// TIA Portal V16 export
// export: Created 2024-09-05T17:39:11.9932458Z, ExportSetting WithDefaults, DisplayName Totally Integrated Automation Portal, DisplayVersion V16 Update 6, DisplayName TIA Portal Version Control Interface, DisplayVersion V16 Update 2, DisplayName TIA Portal Openness, DisplayVersion V16 Update 6, DisplayName STEP 7 Professional, DisplayVersion V16 Update 6, DisplayName STEP 7 Safety, DisplayVersion V16, DisplayName WinCC Advanced, DisplayVersion V16 Update 6
DATA_BLOCK "ServoMain_DB"   // DB6
VERSION : 0.1
// stored: AutoNumber true, DBAccessibleFromOPCUA true, InstanceOfName ServoMain, InstanceOfType FB
"ServoMain"
   // VAR
   //    "TO_BasicPos_TA1-3MA_Instance" { S7_SetPoint := 'True'} : TO_BasicPos;
   //    IEC_Timer_0_Instance { S7_SetPoint := 'True'} : TON_TIME;
   //    "ServoControl_TA1-3MA_Instance" { S7_SetPoint := 'True'} : "ServoControl";
   //    IEC_Timer_0_Instance_1 { S7_SetPoint := 'True'} : TP_TIME;
   // END_VAR
BEGIN
END_DATA_BLOCK
